PROGRAM MAIN
VAR
	nValueInt 	: INT;
	nValueDword : DWORD;
	fValueReal 	: REAL;
	
	sRecipe 	: STRING;
END_VAR

END_PROGRAM

(* stored: Version 1.1.0.1, ProductVersion 3.1.4020.12
   POU MAIN: Id {d09a3875-155e-4b0a-83fc-897e93d6a041}, SpecialFunc None *)
